{attribute addProperty BoxType "EK1960-0000-0021"}
{attribute addProperty Id "FSOEAT %I*FSOE_320A0AF812015"}
{attribute addProperty CRC "2448878193"}
{attribute addProperty SizeInBites "120"}
{attribute addProperty SizeInBytes "15"}
TYPE FSoE_Inputs_91F6EA71 :
STRUCT
	{attribute addProperty Name "FSOE"}
	FSOE AT %I* : FSOE_320A0AF8;
END_STRUCT
END_TYPE

(* stored: Version 1.2.0.0, ProductVersion 3.1.4024.9
   DUT FSoE_Inputs_91F6EA71: Id {3e98408d-ec54-4818-bbdb-f26239e90a5c} *)
